PROGRAM MAIN
VAR
END_VAR

progHSVCntrl();
progFCVCntrl();
progLITCntrl();
progPITCntrl();
progSCACntrl();

END_PROGRAM

(* stored: Version 1.1.0.1, ProductVersion 3.1.4022.17
   POU MAIN: Id {7f5eb3b9-26dd-444a-95ba-4c2038c9772f}, SpecialFunc None *)
